(* IEC 61131-3 sources: plc-home-automation/home_automation/lighting_heating_updated/src/utils/globals, 1 file *)

(* ---- UtilsGlobals.st ---- *)
VAR_GLOBAL CONSTANT

END_VAR

VAR_GLOBAL

  // Global control
  CURRENT_TIME : TIME := T#00:00:00; // Will be updated in WateringControl()
  EXTERNAL_AVERAGE_TEMPERATURE : REAL := 15;  // Will be updated in ExternalAverageTemperature()

END_VAR
